// TIA Portal V20 export
FUNCTION_BLOCK "FB_Pos16_IO"   // FB30142, LAD
{ S7_Optimized_Access := 'TRUE' }
// stored: AutoNumber false, MemoryReserve 100, SetENOAutomatically false
   VAR_INPUT
      Opmode { ExternalAccessible := 'False'; ExternalVisible := 'False'; ExternalWritable := 'False'} : "OPMODE_OUT_UDT";
      TO_PosAxis : TO_PositioningAxis;
      I_iNum_Abspos : Int;
      I_bMan_Enable : Bool;
      I_SS_bHome : Bool;   // 原点传感器
      I_SS_bFW : Bool := TRUE;   // 前限位
      I_SS_bBW : Bool := TRUE;   // 后限位
      I_CMD_bEnableAxis : Bool;   // 使能
      I_CMD_bResetAxis : Bool;   // 复位
      I_CMD_bjogForward : Bool;   // Taster Aufwärts / 正点
      I_CMD_bjogBackward : Bool;   // Taster Abwärts / 反点
      I_CMD_bmoveVelocity : Bool;   // 速度运行
      I_CMD_bstop : Bool;   // 停止
      I_CMD_bfastStop : Bool;   // 急停
      I_CMD_bHoming : Bool;   // 回零
      I_CMD_bGoToPos : Array[0..15] of Bool;   // Start Aufwärts in Automatik / 16个定位
      I_CMD_iGoToPos : Word;   // 16个定位 Word
      I_CMD_bCallAbsPos : Bool;   // 定位位置切换时，单独的定位按钮
      I_CMD_bRelPos : Bool;   // 相对定位
      I_InLock_bEnableAxis : Bool;   // 使能
      I_InLock_bResetAxis : Bool;   // 复位
      I_InLock_bjogForward : Bool;   // Taster Aufwärts / 正点
      I_InLock_bjogBackward : Bool;   // Taster Abwärts / 反点
      I_InLock_bmoveVelocity : Bool;   // 速度运行
      I_InLock_bstop : Bool;   // 停止
      I_InLock_bfastStop : Bool;   // 急停
      I_InLock_bHoming : Bool;   // 回零
      I_InLock_bGoToPos : Array[0..16] of Bool;   // Start Aufwärts in Automatik / 16个定位
      I_InLock_iGoToPos : Word;   // 16个定位 Word
      I_InLock_bCallAbsPos : Bool;   // 定位位置切换时，单独的定位按钮
      I_InLock_bRelPos : Bool;   // 相对定位
      I_InLock_MyBool : Array[0..5] of Bool;   // 临时变量
      I_HMI_bEnableAxis : Bool;   // 使能
      I_HMI_bResetAxis : Bool;   // 复位
      I_HMI_bjogForward : Bool;   // Taster Aufwärts / 正点
      I_HMI_bjogBackward : Bool;   // Taster Abwärts / 反点
      I_HMI_bmoveVelocity : Bool;   // 速度运行
      I_HMI_bstop : Bool;   // 停止
      I_HMI_bfastStop : Bool;   // 急停
      I_HMI_bHoming : Bool;   // 回零
      I_HMI_bGoToPos : Array[0..16] of Bool;   // Start Aufwärts in Automatik / 16个定位
      I_HMI_iGoToPos : Word;   // 16个定位 Word
      I_HMI_bCallAbsPos : Bool;   // 定位位置切换时，单独的定位按钮
      I_HMI_bRelPos : Bool;   // 相对定位
      I_HMI_MyBool : Array[0..5] of Bool;   // 临时变量
      I_CMD_bGoToPos_0 : Bool;   // Start Aufwärts in Automatik / 16个定位自动
      I_InLock_bGoToPos_0 : Bool;   // Start Aufwärts in Automatik / 16个定位条件
      I_HMI_bGoToPos_0 : Bool;   // Start Aufwärts in Automatik / 16个定位HMI
      I_CMD_bGoToPos_1 : Bool;   // Start Aufwärts in Automatik / 16个定位自动
      I_InLock_bGoToPos_1 : Bool;   // Start Aufwärts in Automatik / 16个定位条件
      I_HMI_bGoToPos_1 : Bool;   // Start Aufwärts in Automatik / 16个定位HMI
      I_CMD_bGoToPos_2 : Bool;   // Start Aufwärts in Automatik / 16个定位自动
      I_InLock_bGoToPos_2 : Bool;   // Start Aufwärts in Automatik / 16个定位条件
      I_HMI_bGoToPos_2 : Bool;   // Start Aufwärts in Automatik / 16个定位HMI
      I_CMD_bGoToPos_3 : Bool;   // Start Aufwärts in Automatik / 16个定位自动
      I_InLock_bGoToPos_3 : Bool;   // Start Aufwärts in Automatik / 16个定位条件
      I_HMI_bGoToPos_3 : Bool;   // Start Aufwärts in Automatik / 16个定位HMI
      I_CMD_bGoToPos_4 : Bool;   // Start Aufwärts in Automatik / 16个定位自动
      I_InLock_bGoToPos_4 : Bool;   // Start Aufwärts in Automatik / 16个定位条件
      I_HMI_bGoToPos_4 : Bool;   // Start Aufwärts in Automatik / 16个定位HMI
      I_CMD_bGoToPos_5 : Bool;   // Start Aufwärts in Automatik / 16个定位自动
      I_InLock_bGoToPos_5 : Bool;   // Start Aufwärts in Automatik / 16个定位条件
      I_HMI_bGoToPos_5 : Bool;   // Start Aufwärts in Automatik / 16个定位HMI
      I_CMD_bGoToPos_6 : Bool;   // Start Aufwärts in Automatik / 16个定位自动
      I_InLock_bGoToPos_6 : Bool;   // Start Aufwärts in Automatik / 16个定位条件
      I_HMI_bGoToPos_6 : Bool;   // Start Aufwärts in Automatik / 16个定位HMI
      I_CMD_bGoToPos_7 : Bool;   // Start Aufwärts in Automatik / 16个定位自动
      I_InLock_bGoToPos_7 : Bool;   // Start Aufwärts in Automatik / 16个定位条件
      I_HMI_bGoToPos_7 : Bool;   // Start Aufwärts in Automatik / 16个定位HMI
      I_CMD_bGoToPos_8 : Bool;   // Start Aufwärts in Automatik / 16个定位自动
      I_InLock_bGoToPos_8 : Bool;   // Start Aufwärts in Automatik / 16个定位条件
      I_HMI_bGoToPos_8 : Bool;   // Start Aufwärts in Automatik / 16个定位HMI
      I_iHomeMode : Int := 3;
   END_VAR
   VAR_OUTPUT
      O_Status_bAxisReady : Bool;   // 轴通讯正常
      O_Status_bAxisEnabled : Bool;   // 轴使能
      O_Status_bjogForward : Bool;   // 轴正点中
      O_Status_bjogBackward : Bool;   // 轴反点中
      O_Status_bHomed : Bool;   // 轴归零完成
      O_Status_bAtHome : Bool;   // 轴在零位
      O_Status_bSstill : Bool;   // 轴静止
      O_Status_bAxisBusy : Bool;   // 轴运行中
      O_Status_bAxisSyned : Bool;   // 同步上
      O_Status_bAxisError : Bool;   // 轴报警
      O_Status_bAtPos : Array[0..15] of Bool;   // Ausgang Aufwärts / 在目标位置上
      O_Status_bPosDone : Array[0..15] of Bool;   // 定位完成
      O_Status_bPosing : Array[0..15] of Bool;   // Ausgang Aufwärts / 定位中
      O_Status_bRelPosDone : Bool;   // 相对定位完成
      O_Status_rActPos : LReal;   // 实际位置
      O_Status_rActSpeed : LReal;   // 实际速度
      O_Status_iAxisFaultNum : UDInt;   // 轴报警代码
      O_Status_iDriveFaultNum : UDInt;   // 驱动报警代码
      O_Status_iFBStatus : Word;   // 运动功能块状态
      O_Status_iMCStatus : Word;   // 运动指令状态
      O_Status_rDriveTorque : LReal;   // 驱动扭矩
      O_Status_rDriveTemp : LReal;   // 驱动温度
      O_Status_rDriveRpm : LReal;   // 驱动转速
      O_Status_AxisName : WString[24] := WSTRING#'No axis';   // Name of axis
      O_Status_mybool : Array[0..5] of Bool;   // 备用
      O_Status_myLreal : Array[0..5] of LReal;   // 备用
   END_VAR
   VAR_IN_OUT
      I_Para_rJog_Speed : Array[0..2] of LReal;   // 点动速度/ACC/DEC/JERK
      I_Para_rMV_Speed : Array[0..2] of LReal;   // 速度运行速度/ACC/DEC/JERK
      I_Para_rStop_Dec : Array[0..1] of LReal;   // 速度运行速度/ACC/DEC/JERK
      I_Para_rEStop_Dec : Array[0..1] of LReal;   // 速度运行速度/ACC/DEC/JERK
      I_Para_iNum_Abspos : Int := 4;
      I_Para_rPos_Abs : Array[0..16] of LReal;   // 绝对定位目标位置 / Over travel switch set
      I_Para_rSpeed_Abs : Array[0..16] of LReal;   // Endlage Unten / 绝对定位速度
      I_Para_rAcc_Set : Array[0..16] of LReal;   // 绝对定位加速度 / Overtravel switch Reset
      I_Para_rDec_Set : Array[0..16] of LReal;   // 绝对定位减速度 / Belt check sensor
      I_Para_rJerk_Set : Array[0..16] of LReal;   // 绝对定位加加速度
      I_Para_rSpeedPercent : LReal := 20.0;   // Endlage Unten / 速度设定百分比
   END_VAR
   VAR
      instAxis01 { ExternalAccessible := 'False'; ExternalVisible := 'False'; ExternalWritable := 'False'} : "LAxisCtrl_PosAxis";
      instShearAxisStatus { S7_SetPoint := 'True'} : "LAxisCtrl_GetAxisStatusWord";
      RT_Reset { S7_SetPoint := 'True'} : R_TRIG;
      RT_PB { ExternalAccessible := 'False'; ExternalVisible := 'False'; ExternalWritable := 'False'} : Array[0..19] of R_TRIG;   // Störungen / Alarms
      FT_PB { ExternalAccessible := 'False'; ExternalVisible := 'False'; ExternalWritable := 'False'; S7_SetPoint := 'True'} : Array[0..19] of F_TRIG;   // Störungen unterdrücken, Belegung identisch mit "Alarm" / Hide Alarms, identical with "Alarm"
      TON_PB { ExternalAccessible := 'False'; ExternalVisible := 'False'; ExternalWritable := 'False'} : Array[0..19] of TON_TIME;   // Fallende Flanke / Falling edge
      TOF_PB { ExternalAccessible := 'False'; ExternalVisible := 'False'; ExternalWritable := 'False'} : Array[0..19] of TOF_TIME;   // Negativer Impuls / Negative pulse
      i { S7_SetPoint := 'True'} : Int;
      temp_cmd_bEnableAxis { ExternalAccessible := 'False'; ExternalVisible := 'False'; ExternalWritable := 'False'} : Bool;
      temp_cmd_bresetAxis { ExternalAccessible := 'False'; ExternalVisible := 'False'; ExternalWritable := 'False'} : Bool;
      temp_cmd_bjogForward { ExternalAccessible := 'False'; ExternalVisible := 'False'; ExternalWritable := 'False'} : Bool;
      temp_cmd_bjogBackward { ExternalAccessible := 'False'; ExternalVisible := 'False'; ExternalWritable := 'False'} : Bool;
      temp_cmd_bmoveVelocity { ExternalAccessible := 'False'; ExternalVisible := 'False'; ExternalWritable := 'False'} : Bool;
      temp_cmd_bstop { ExternalAccessible := 'False'; ExternalVisible := 'False'; ExternalWritable := 'False'} : Bool;
      temp_cmd_bfastStop { ExternalAccessible := 'False'; ExternalVisible := 'False'; ExternalWritable := 'False'} : Bool;
      temp_cmd_bhoming { ExternalAccessible := 'False'; ExternalVisible := 'False'; ExternalWritable := 'False'} : Bool;
      temp_cmd_bGoToPos { ExternalAccessible := 'False'; ExternalVisible := 'False'; ExternalWritable := 'False'} : Array[0..16] of Bool;
      temp_cmd_iGoToPos : Word;
      temp_cmd_bCallAbsPos : Bool;
      temp_cmd_bRelPos : Bool;
      temp_Para_rJog_Speed { ExternalAccessible := 'False'; ExternalVisible := 'False'; ExternalWritable := 'False'} : LReal;
      temp_configuration { ExternalAccessible := 'False'; ExternalVisible := 'False'; ExternalWritable := 'False'} : "LAxisCtrl_typeAxisConfig";   // Diagnostics structure
      temp_Status { ExternalAccessible := 'False'; ExternalVisible := 'False'; ExternalWritable := 'False'} : Word;
      temp_AxisEnabled { ExternalAccessible := 'False'; ExternalVisible := 'False'; ExternalWritable := 'False'} : Bool;
      temp_CommandBusy { ExternalAccessible := 'False'; ExternalVisible := 'False'; ExternalWritable := 'False'} : Bool;
      temp_CommandDone { ExternalAccessible := 'False'; ExternalVisible := 'False'; ExternalWritable := 'False'} : Bool;
      temp_CommandAborted { ExternalAccessible := 'False'; ExternalVisible := 'False'; ExternalWritable := 'False'} : Bool;
      temp_InVelocity { ExternalAccessible := 'False'; ExternalVisible := 'False'; ExternalWritable := 'False'} : Bool;
      temp_jogSelected { ExternalAccessible := 'False'; ExternalVisible := 'False'; ExternalWritable := 'False'} : Bool;
      tempPosAbsoluteSelected { ExternalAccessible := 'False'; ExternalVisible := 'False'; ExternalWritable := 'False'} : Bool;
      temp_diagnostics { ExternalAccessible := 'False'; ExternalVisible := 'False'; ExternalWritable := 'False'} : "LAxisCtrl_typeDiagnostics";
      temp_stop_Dec { ExternalAccessible := 'False'; ExternalVisible := 'False'; ExternalWritable := 'False'} : LReal;
      temp_faststop_Dec { ExternalAccessible := 'False'; ExternalVisible := 'False'; ExternalWritable := 'False'} : LReal;
      temp_cmd_bGoToPosAll : Bool;
      temp_iFBStatus : Word;
      temp_iMCStatus : Word;
      old_iFBStatus : Word;
      old_iMCStatus : Word;
   END_VAR
BEGIN

REGION Network 1
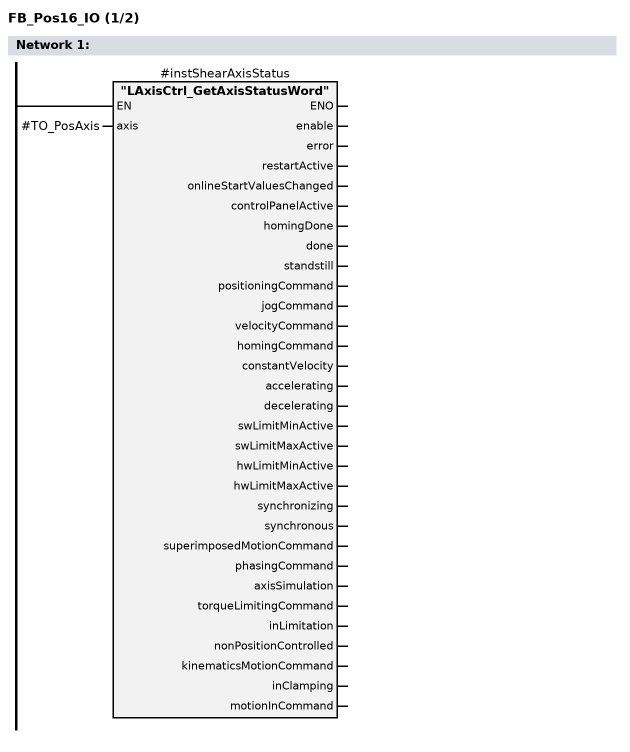
   RUNG wire#powerrail
      #instShearAxisStatus(axis := #TO_PosAxis, enable =>, error =>, restartActive =>, onlineStartValuesChanged =>, controlPanelActive =>, homingDone =>, done =>, standstill =>, positioningCommand =>, jogCommand =>, velocityCommand =>, homingCommand =>, constantVelocity =>, accelerating =>, decelerating =>, swLimitMinActive =>, swLimitMaxActive =>, hwLimitMinActive =>, hwLimitMaxActive =>, synchronizing =>, synchronous =>, superimposedMotionCommand =>, phasingCommand =>, axisSimulation =>, torqueLimitingCommand =>, inLimitation =>, nonPositionControlled =>, kinematicsMotionCommand =>, inClamping =>, motionInCommand =>)
   END_RUNG
   // the same network as SCL:
   #instShearAxisStatus(axis := #TO_PosAxis);   // "LAxisCtrl_GetAxisStatusWord"
END_REGION

REGION Network 2: LAxisCtrl
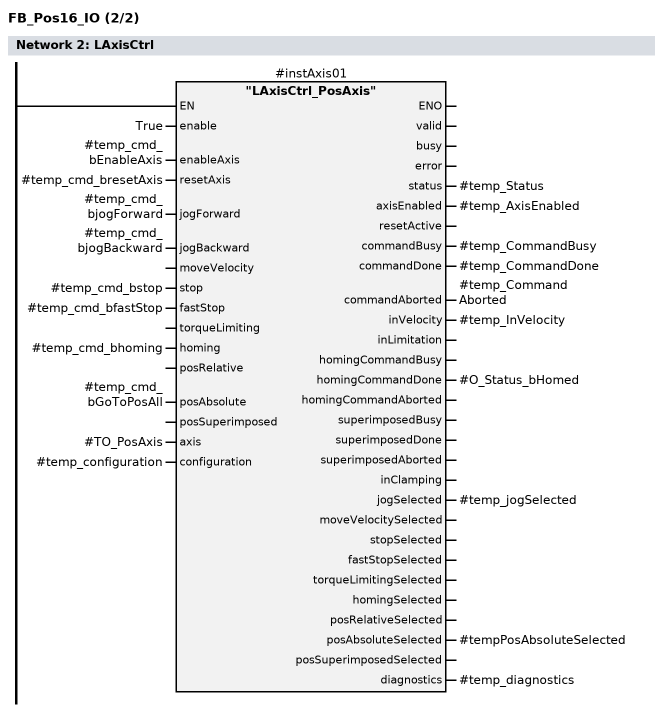
   RUNG wire#powerrail
      #instAxis01(enable := True, enableAxis := #temp_cmd_bEnableAxis, resetAxis := #temp_cmd_bresetAxis, jogForward := #temp_cmd_bjogForward, jogBackward := #temp_cmd_bjogBackward, moveVelocity :=, stop := #temp_cmd_bstop, fastStop := #temp_cmd_bfastStop, torqueLimiting :=, homing := #temp_cmd_bhoming, posRelative :=, posAbsolute := #temp_cmd_bGoToPosAll, posSuperimposed :=, axis := #TO_PosAxis, configuration := #temp_configuration, valid =>, busy =>, error =>, status => #temp_Status, axisEnabled => #temp_AxisEnabled, resetActive =>, commandBusy => #temp_CommandBusy, commandDone => #temp_CommandDone, commandAborted => #temp_CommandAborted, inVelocity => #temp_InVelocity, inLimitation =>, homingCommandBusy =>, homingCommandDone => #O_Status_bHomed, homingCommandAborted =>, superimposedBusy =>, superimposedDone =>, superimposedAborted =>, inClamping =>, jogSelected => #temp_jogSelected, moveVelocitySelected =>, stopSelected =>, fastStopSelected =>, torqueLimitingSelected =>, homingSelected =>, posRelativeSelected =>, posAbsoluteSelected => #tempPosAbsoluteSelected, posSuperimposedSelected =>, diagnostics => #temp_diagnostics)
   END_RUNG
   // the same network as SCL:
   #instAxis01(enable := True,   // "LAxisCtrl_PosAxis"
               enableAxis := #temp_cmd_bEnableAxis,
               resetAxis := #temp_cmd_bresetAxis,
               jogForward := #temp_cmd_bjogForward,
               jogBackward := #temp_cmd_bjogBackward,
               stop := #temp_cmd_bstop,
               fastStop := #temp_cmd_bfastStop,
               homing := #temp_cmd_bhoming,
               posAbsolute := #temp_cmd_bGoToPosAll,
               axis := #TO_PosAxis,
               configuration := #temp_configuration,
               status => #temp_Status,
               axisEnabled => #temp_AxisEnabled,
               commandBusy => #temp_CommandBusy,
               commandDone => #temp_CommandDone,
               commandAborted => #temp_CommandAborted,
               inVelocity => #temp_InVelocity,
               homingCommandDone => #O_Status_bHomed,
               jogSelected => #temp_jogSelected,
               posAbsoluteSelected => #tempPosAbsoluteSelected,
               diagnostics => #temp_diagnostics);
END_REGION

REGION Network 3 (SCL): input
   #temp_cmd_bEnableAxis  := #I_CMD_bEnableAxis OR (#I_HMI_bEnableAxis AND #I_bMan_Enable);
   #temp_cmd_bresetAxis   := #I_CMD_bResetAxis;
   #temp_cmd_bjogForward  := #I_InLock_bjogForward AND (#I_CMD_bjogForward OR (#I_HMI_bjogForward AND #I_bMan_Enable));
   #temp_cmd_bjogBackward := #I_InLock_bjogBackward AND (#I_CMD_bjogBackward OR (#I_HMI_bjogBackward AND #I_bMan_Enable));
   #temp_cmd_bstop        := #I_CMD_bstop OR (#I_HMI_bstop AND #I_bMan_Enable);
   #temp_cmd_bfastStop    := #I_CMD_bfastStop;
   #temp_cmd_bhoming      := #I_InLock_bHoming AND (#I_CMD_bHoming OR #I_HMI_bHoming);
END_REGION

REGION Network 4 (SCL): Configuration
   //#I_Para_rJog_Speed[0] := 10.0;
   #I_Para_rMV_Speed[0]  := 10.0;
   #I_Para_rStop_Dec[0]  := 20.0;
   #I_Para_rEStop_Dec[0] := 50.0;

   #I_Para_rJog_Speed[1] := 10.0 * #I_Para_rJog_Speed[0];
   #I_Para_rJog_Speed[2] := 10.0 * #I_Para_rJog_Speed[0];
   #I_Para_rMV_Speed[1] := 10.0 * #I_Para_rMV_Speed[0];
   #I_Para_rMV_Speed[2] := 10.0 * #I_Para_rMV_Speed[0];
   #I_Para_rStop_Dec[1] := 100.0 * #I_Para_rStop_Dec[0];
   #I_Para_rEStop_Dec[1] := 100.0 * #I_Para_rEStop_Dec[0];

   IF #temp_configuration.jog.velocity <> #I_Para_rJog_Speed[0] OR
       #temp_configuration.jog.acceleration <> #I_Para_rJog_Speed[1] OR
       #temp_configuration.jog.deceleration <> #I_Para_rJog_Speed[2] OR
       #temp_configuration.moveVelocity.acceleration <> #I_Para_rMV_Speed[0] OR
       #temp_configuration.moveVelocity.deceleration <> #I_Para_rMV_Speed[1] OR
       #temp_configuration.moveVelocity.acceleration <> #I_Para_rMV_Speed[2] OR
       #temp_configuration.stop.deceleration <> #I_Para_rStop_Dec[0] OR
       #temp_configuration.stop.jerk <> #I_Para_rStop_Dec[1] OR
       #temp_configuration.fastStop.deceleration <> #I_Para_rEStop_Dec[0] OR
       #temp_configuration.fastStop.jerk <> #I_Para_rEStop_Dec[1]
   THEN
       // Jog
       #temp_configuration.jog.velocity := #I_Para_rJog_Speed[0];
       #temp_configuration.jog.acceleration := #I_Para_rJog_Speed[1];
       #temp_configuration.jog.deceleration := #I_Para_rJog_Speed[2];
       // Move
       #temp_configuration.moveVelocity.velocity := #I_Para_rMV_Speed[0];
       #temp_configuration.moveVelocity.acceleration := #I_Para_rMV_Speed[1];
       #temp_configuration.moveVelocity.deceleration := #I_Para_rMV_Speed[2];
       // Stop   
       #temp_configuration.stop.deceleration := #I_Para_rStop_Dec[0];
       #temp_configuration.stop.jerk := #I_Para_rStop_Dec[1];
       //faststoo
       #temp_configuration.fastStop.deceleration := #I_Para_rEStop_Dec[0];
       #temp_configuration.fastStop.jerk := #I_Para_rEStop_Dec[1];
   END_IF;

   // Homing
   #temp_configuration.homing.mode := #I_iHomeMode;//I_iHomeMode
   #temp_configuration.homing.position := 0;//I_iHomePos

   //abspos
   FOR #i := 1 TO 16 DO
       #I_Para_rAcc_Set[#i] := 10.0 * #I_Para_rSpeed_Abs[0];
       #I_Para_rDec_Set[#i] := 10.0 * #I_Para_rSpeed_Abs[0];
       #I_Para_rJerk_Set[#i] := 100.0 * #I_Para_rSpeed_Abs[0];
   END_FOR;


   //#temp_posAbsolute := (I_CMD_iGoToPos <> 16#0);
   #temp_cmd_bGoToPos[1] := (((#Opmode.Automatic_active=1 OR #Opmode.SingleStep_active=1) AND #I_CMD_iGoToPos = 1) OR (#Opmode.Manual_active AND  #I_HMI_iGoToPos = 1)) AND #I_InLock_bGoToPos[1];
   #temp_cmd_bGoToPos[2] := (((#Opmode.Automatic_active=1 OR #Opmode.SingleStep_active=1) AND #I_CMD_iGoToPos = 2) OR (#Opmode.Manual_active AND  #I_HMI_iGoToPos = 2)) AND #I_InLock_bGoToPos[2];
   #temp_cmd_bGoToPos[3] := (((#Opmode.Automatic_active=1 OR #Opmode.SingleStep_active=1) AND #I_CMD_iGoToPos = 3) OR (#Opmode.Manual_active AND  #I_HMI_iGoToPos = 3)) AND #I_InLock_bGoToPos[3];
   #temp_cmd_bGoToPos[4] := (((#Opmode.Automatic_active=1 OR #Opmode.SingleStep_active=1) AND #I_CMD_iGoToPos = 4) OR (#Opmode.Manual_active AND  #I_HMI_iGoToPos = 4)) AND #I_InLock_bGoToPos[4];
   #temp_cmd_bGoToPos[5] := (((#Opmode.Automatic_active=1 OR #Opmode.SingleStep_active=1) AND #I_CMD_iGoToPos = 5) OR (#Opmode.Manual_active AND  #I_HMI_iGoToPos = 5)) AND #I_InLock_bGoToPos[5];
   #temp_cmd_bGoToPos[6] := (((#Opmode.Automatic_active=1 OR #Opmode.SingleStep_active=1) AND #I_CMD_iGoToPos = 6) OR (#Opmode.Manual_active AND  #I_HMI_iGoToPos = 6)) AND #I_InLock_bGoToPos[6];
   #temp_cmd_bGoToPos[7] := (((#Opmode.Automatic_active=1 OR #Opmode.SingleStep_active=1) AND #I_CMD_iGoToPos = 7) OR (#Opmode.Manual_active AND  #I_HMI_iGoToPos = 7)) AND #I_InLock_bGoToPos[7];
   #temp_cmd_bGoToPos[8] := (((#Opmode.Automatic_active=1 OR #Opmode.SingleStep_active=1) AND #I_CMD_iGoToPos = 8) OR (#Opmode.Manual_active AND  #I_HMI_iGoToPos = 8)) AND #I_InLock_bGoToPos[8];
   #temp_cmd_bGoToPos[9] := (((#Opmode.Automatic_active=1 OR #Opmode.SingleStep_active=1) AND #I_CMD_iGoToPos = 9) OR (#Opmode.Manual_active AND  #I_HMI_iGoToPos = 9)) AND #I_InLock_bGoToPos[9];
   #temp_cmd_bGoToPos[10] := (((#Opmode.Automatic_active=1 OR #Opmode.SingleStep_active=1) AND #I_CMD_iGoToPos = 10) OR (#Opmode.Manual_active AND  #I_HMI_iGoToPos = 10)) AND #I_InLock_bGoToPos[10];
   #temp_cmd_bGoToPos[11] := (((#Opmode.Automatic_active=1 OR #Opmode.SingleStep_active=1) AND #I_CMD_iGoToPos = 11) OR (#Opmode.Manual_active AND  #I_HMI_iGoToPos = 11)) AND #I_InLock_bGoToPos[11];
   #temp_cmd_bGoToPos[12] := (((#Opmode.Automatic_active=1 OR #Opmode.SingleStep_active=1) AND #I_CMD_iGoToPos = 12) OR (#Opmode.Manual_active AND  #I_HMI_iGoToPos = 12)) AND #I_InLock_bGoToPos[12];
   #temp_cmd_bGoToPos[13] := (((#Opmode.Automatic_active=1 OR #Opmode.SingleStep_active=1) AND #I_CMD_iGoToPos = 13) OR (#Opmode.Manual_active AND  #I_HMI_iGoToPos = 13)) AND #I_InLock_bGoToPos[13];
   #temp_cmd_bGoToPos[14] := (((#Opmode.Automatic_active=1 OR #Opmode.SingleStep_active=1) AND #I_CMD_iGoToPos = 14) OR (#Opmode.Manual_active AND  #I_HMI_iGoToPos = 14)) AND #I_InLock_bGoToPos[14];
   #temp_cmd_bGoToPos[15] := (((#Opmode.Automatic_active=1 OR #Opmode.SingleStep_active=1) AND #I_CMD_iGoToPos = 15) OR (#Opmode.Manual_active AND  #I_HMI_iGoToPos = 15)) AND #I_InLock_bGoToPos[15];
   #temp_cmd_bGoToPos[16] := (((#Opmode.Automatic_active=1 OR #Opmode.SingleStep_active=1) AND #I_CMD_iGoToPos = 16) OR (#Opmode.Manual_active AND  #I_HMI_iGoToPos = 16)) AND #I_InLock_bGoToPos[16];

   #temp_cmd_bGoToPosAll := #temp_cmd_bGoToPos[1] OR #temp_cmd_bGoToPos[2] OR #temp_cmd_bGoToPos[3] OR #temp_cmd_bGoToPos[4]
   OR #temp_cmd_bGoToPos[5] OR #temp_cmd_bGoToPos[6] OR #temp_cmd_bGoToPos[7] OR #temp_cmd_bGoToPos[8]
   OR #temp_cmd_bGoToPos[9] OR #temp_cmd_bGoToPos[10] OR #temp_cmd_bGoToPos[11] OR #temp_cmd_bGoToPos[12]
   OR #temp_cmd_bGoToPos[13] OR #temp_cmd_bGoToPos[14] OR #temp_cmd_bGoToPos[15] OR #temp_cmd_bGoToPos[16]
   ;
   //#temp_posAbsolute :=
   //I_bGoToPos[0] OR I_bGoToPos[1] OR I_bGoToPos[2] OR I_bGoToPos[3] OR
   //I_bGoToPos[4] OR I_bGoToPos[5] OR I_bGoToPos[6] OR I_bGoToPos[7] OR
   //I_bGoToPos[8] OR I_bGoToPos[9] OR I_bGoToPos[10] OR I_bGoToPos[11] OR
   //I_bGoToPos[12] OR I_bGoToPos[13] OR I_bGoToPos[14] OR I_bGoToPos[15];

   FOR #i := 1 TO 16 DO
   //    #RT_PB[#i](CLK := I_bGoToPos[#i]);
       #RT_PB[#i](CLK := #temp_cmd_bGoToPos[#i]);

       IF #RT_PB[#i].Q THEN
           #temp_configuration.posAbsolute.position := #I_Para_rPos_Abs[#i];
           #temp_configuration.posAbsolute.velocity := #I_Para_rSpeed_Abs[#i];
           #temp_configuration.posAbsolute.direction := 3;//temp_posAbsolute_direction

           #temp_configuration.posAbsolute.acceleration := #I_Para_rAcc_Set[#i];
           #temp_configuration.posAbsolute.deceleration := #I_Para_rDec_Set[#i];
           #temp_configuration.posAbsolute.jerk := #I_Para_rJerk_Set[#i];

       END_IF;
   END_FOR;
END_REGION

REGION Network 5 (SCL): output
   #O_Status_bAxisReady := true;//#TO_PosAxis.StatusWord.%X1;
   #O_Status_bAxisEnabled := #temp_AxisEnabled;
   #O_Status_bjogForward := #temp_cmd_bjogForward;// AND #temp_jogSelected;
   #O_Status_bjogBackward := #temp_cmd_bjogBackward;// AND #temp_jogSelected;
   //#O_Status_bHomed := #TO_PosAxis.StatusWord.%X5;
   #O_Status_bAxisError := #TO_PosAxis.StatusWord.%X1;
   #O_Status_rActPos := #TO_PosAxis.ActualPosition;
   #O_Status_rActSpeed := #TO_PosAxis.ActualVelocity;
   #O_Status_iAxisFaultNum := #TO_PosAxis.ErrorDetail.Number;
   //O_DriveFaultNum
   //O_Status_iFBStatus := #temp_diagnostics.status;
   //O_Status_iMCStatus := #temp_diagnostics.subfunctionStatus;
   //O_Torque
   //oAxisName  := 

   FOR #i := 0 TO 15 DO
       #O_Status_bAtPos[#i] := "FC_bNearIn"(rAct := #O_Status_rActPos, rTgt := #I_Para_rPos_Abs[#i], rDelta := 1.0, bModule := 0, rModulo := 0);
   END_FOR;

   //O_bPosDone
   //O_bPosing
   //#tempPosAbsoluteSelected
END_REGION

REGION Network 6 (SCL): Reset
   #RT_Reset(CLK := #temp_cmd_bresetAxis);
   IF #RT_Reset.Q THEN
       #O_Status_iFBStatus := 16#00;
       #O_Status_iMCStatus := 16#00;
   END_IF;

   #temp_iFBStatus := #temp_diagnostics.status;
   IF #temp_iFBStatus <> #old_iFBStatus THEN
       #O_Status_iFBStatus := #temp_diagnostics.status;
       #old_iFBStatus := #temp_iFBStatus;
   END_IF;
   #temp_iMCStatus := #temp_diagnostics.subfunctionStatus;
   IF #temp_iMCStatus <> #old_iMCStatus THEN
       #O_Status_iFBStatus := #temp_diagnostics.subfunctionStatus;
       #old_iMCStatus := #temp_iMCStatus;
   END_IF;
END_REGION

REGION Network 7 (SCL)
   (*
   FOR #i := 9 TO 16 DO
       IF #I_iNum_Abspos < #i THEN
           I_InLock_bGoToPos[#i] := false;
       END_IF;
   END_FOR;
   *)
END_REGION
END_FUNCTION_BLOCK
